(* 
	FB_MoveAbsolute: Controls absolute movement using target position, velocity, acceleration, and deceleration. 
*)
FUNCTION_BLOCK FB_MoveAbsolute 
VAR_INPUT
	fTargetPosition 	: REAL;
	fTargetVelocity 	: REAL; 
	fAccMax 			: REAL; 
	fDecMax 			: REAL;	
	fTolerance			: REAL := 1E-6;	
END_VAR

VAR
	_fVelocity 			: REAL;
	_fPosition 			: REAL;
	_bIsReached			: BOOL;
END_VAR

fTargetVelocity := ABS(fTargetVelocity); 
fAccMax := ABS(fAccMax);
fDecMax := -ABS(fDecMax);

IF F_Compare(fTargetPosition, _fPosition, fTolerance) THEN
	_fVelocity := 0;
	_fPosition := fTargetPosition;
	_bIsReached := TRUE;	
ELSE
	(* Calculate velocity and position *)
	IF fTargetPosition > _fPosition THEN		
		IF _fVelocity < 0 THEN
			_fVelocity := MIN(_fVelocity - fDecMax * GVL_Core.fbSystem.fDeltaTime * GVL_Core.fbSystem.fTimeScaling, fTargetVelocity);
		ELSE
			IF _fVelocity > fTargetVelocity THEN
				_fVelocity := MAX(_fVelocity + fDecMax * GVL_Core.fbSystem.fDeltaTime * GVL_Core.fbSystem.fTimeScaling, fTargetVelocity);
			ELSE
				_fVelocity := MIN(_fVelocity + fAccMax * GVL_Core.fbSystem.fDeltaTime * GVL_Core.fbSystem.fTimeScaling, fTargetVelocity);
			END_IF

			_fVelocity := MIN(SQRT((_fPosition - fTargetPosition) * 2.0 * fDecMax - 1.5 * GVL_Core.fbSystem.fDeltaTime * GVL_Core.fbSystem.fTimeScaling * fDecMax), _fVelocity);
		END_IF

		_fPosition := _fPosition + MIN(_fVelocity * GVL_Core.fbSystem.fDeltaTime * GVL_Core.fbSystem.fTimeScaling, fTargetPosition - _fPosition);	
	ELSE		
		IF _fVelocity > 0 THEN
			_fVelocity := MAX(_fVelocity + fDecMax * GVL_Core.fbSystem.fDeltaTime * GVL_Core.fbSystem.fTimeScaling, -fTargetVelocity);
		ELSE
			IF _fVelocity < -fTargetVelocity THEN
				_fVelocity := MIN(_fVelocity - fDecMax * GVL_Core.fbSystem.fDeltaTime * GVL_Core.fbSystem.fTimeScaling, -fTargetVelocity);
			ELSE				
				_fVelocity := MAX(_fVelocity - fAccMax * GVL_Core.fbSystem.fDeltaTime * GVL_Core.fbSystem.fTimeScaling, -fTargetVelocity);
			END_IF
			
			_fVelocity := MAX(-SQRT((_fPosition - fTargetPosition) * 2.0 * -fDecMax - 1.5 * GVL_Core.fbSystem.fDeltaTime * GVL_Core.fbSystem.fTimeScaling * fDecMax), _fVelocity);
	   END_IF

		_fPosition := _fPosition + MAX(_fVelocity * GVL_Core.fbSystem.fDeltaTime * GVL_Core.fbSystem.fTimeScaling, fTargetPosition - _fPosition);	
	END_IF;
	
	_bIsReached := FALSE;		
END_IF;

(*
    Indicates whether the drive has reached its target position.

    This property reflects the internal state of the drive control system.
    It returns TRUE if the drive has achieved the desired position within the specified
    tolerance limits; otherwise, it returns FALSE.
*)
PROPERTY bIsReached : BOOL
GET
bIsReached := THIS^._bIsReached;
END_GET
END_PROPERTY

(*
    Actual Drive Position
	
	The fPosition property provides the current position for the drive.
*)
PROPERTY fPosition : REAL
GET
fPosition := _fPosition;
END_GET
SET
_fPosition := fPosition;
END_SET
END_PROPERTY

(*
    Actual Drive Velocity
	
	The fVelocity property provides the current velocity for the drive.
*)
PROPERTY fVelocity : REAL
GET
fVelocity := _fVelocity;
END_GET
SET
_fVelocity := fVelocity;
END_SET
END_PROPERTY

END_FUNCTION_BLOCK

(* stored: Version 1.1.0.1, ProductVersion 3.1.4024.12
   POU FB_MoveAbsolute: Id {33b9870f-0a9c-08e8-23f5-ccdbe10d56b1}, SpecialFunc None
   Property bIsReached: Id {320d2df9-9e83-0523-347f-f35c1b62f10e}
   Get Get: Id {eacc081e-c993-0ad0-39a3-fb17f6116bc2}
   Property fPosition: Id {a21654d8-2e5f-07b0-0e69-8fa21086f7cb}
   Get Get: Id {c28b23b5-f544-0523-161b-cc1f0434641a}
   Set Set: Id {f7fb7a3c-f492-0b49-0050-c94ddcd18011}
   Property fVelocity: Id {9afbc35c-a683-0626-3ff9-fba8fb0d85b9}
   Get Get: Id {ddc4c959-cefa-0b1a-0065-0f24a9c97365}
   Set Set: Id {a85e303f-e873-0b76-39a2-e99cbc778880} *)
